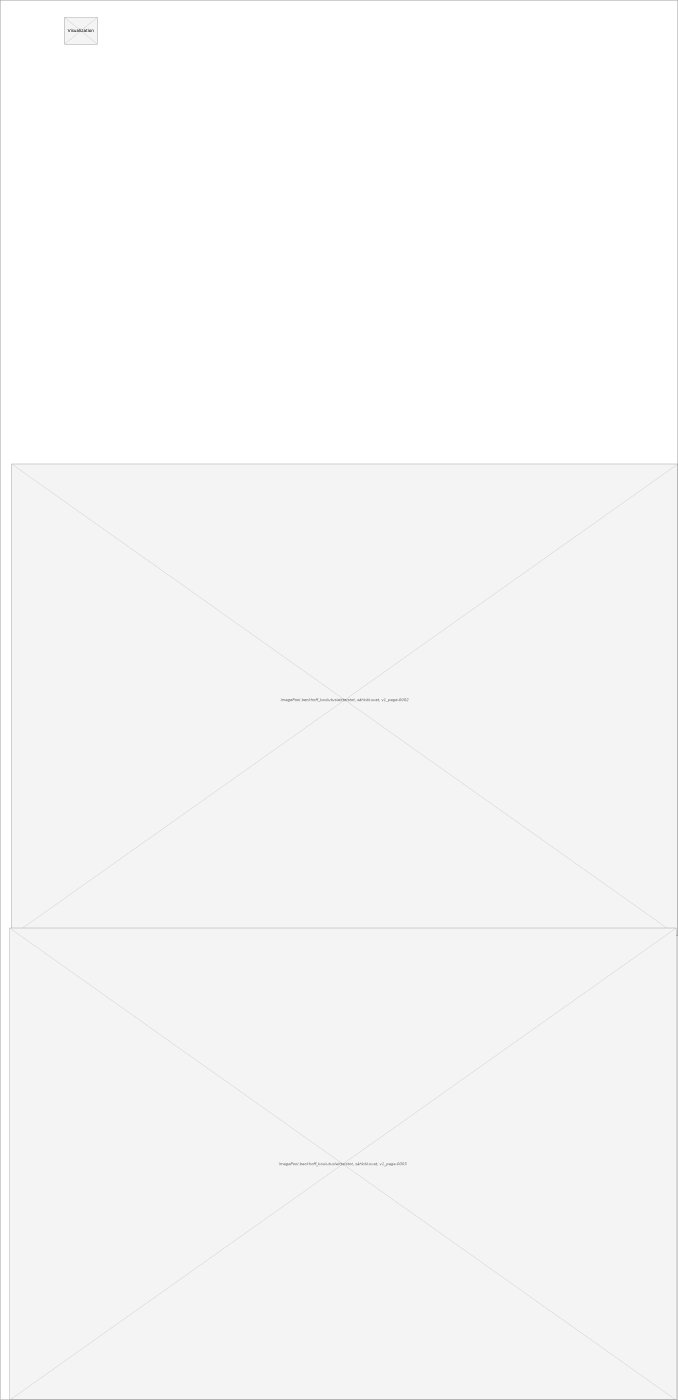
VISUALIZATION Huoltosivu  // 1783x3677, background image ImagePool.beckhoff_koulutuslaitteistot, sähkökuvat, v1_page-0001
    Image (169,45 87x71), "Visualization", image: VisuDialogs.ImagePoolDialogs.FileOpen
        OnMouseClick: change screen: Visualization
    Image (30,1218 1753x1240), image: ImagePool.beckhoff_koulutuslaitteistot, sähkökuvat, v1_page-0002
    Image (25,2437 1753x1240), image: ImagePool.beckhoff_koulutuslaitteistot, sähkökuvat, v1_page-0003
END_VISUALIZATION

(* stored: Version 1.1.0.1, ProductVersion 3.1.4024.11
   Visu Huoltosivu: Id {3cc23ecc-f1b9-415b-b706-34028e665d78} *)
